// TIA Portal V20 export
DATA_BLOCK "ManualOperationControl_U1Em3"   // DB142
// stored: MemoryReserve 100
   VAR
      manualOperationEm { ExternalAccessible := 'False'; ExternalVisible := 'False'; ExternalWritable := 'False'} : "LAF_typeManEm";
      manualOperationEmArea { ExternalAccessible := 'False'; ExternalVisible := 'False'; ExternalWritable := 'False'} : Array[1..2] of "LAF_typeManOperationArea";
      manualOperationCms { ExternalAccessible := 'False'; ExternalVisible := 'False'; ExternalWritable := 'False'} : Array[1..45] of "LAF_typeManOperation";
      axis { ExternalAccessible := 'False'; ExternalVisible := 'False'; ExternalWritable := 'False'} : Array[0..0] of "LBC_typeAxisControlInterface";
      axis64Pos { ExternalAccessible := 'False'; ExternalVisible := 'False'; ExternalWritable := 'False'} : Array[0..0] of "LBC_typeAxis64PosInterface";
      softCam { ExternalAccessible := 'False'; ExternalVisible := 'False'; ExternalWritable := 'False'} : Array[0..0] of "LER_typeSoftCamRelation";
      sina { ExternalAccessible := 'False'; ExternalVisible := 'False'; ExternalWritable := 'False'} : Array[0..0] of "LBC_typeSinaSpeedInterface";
      twoWayActuator { ExternalAccessible := 'False'; ExternalVisible := 'False'; ExternalWritable := 'False'} : Array[0..1] of "LBC_typeTwoWayActuatorInterface";
   END_VAR
BEGIN
   manualOperationEm.equipmentModuleNum := 1040;
END_DATA_BLOCK
